ADAPTER EBBusAdapter
  (* Standard: 61499-1 *)
  (* Version 0.0, 2008-04-22, GE, 4DIAC-Consortium *)
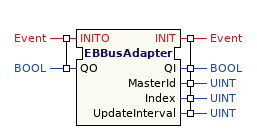
  EVENT_INPUT
    INITO WITH QO; (* Initialization Confirm *)
  END_EVENT
  EVENT_OUTPUT
    INIT WITH Index, UpdateInterval, MasterId, QI; (* Service Initialization *)
  END_EVENT
  VAR_INPUT
    QO : BOOL;
  END_VAR
  VAR_OUTPUT
    QI : BOOL;
    MasterId : UINT;
    Index : UINT;
    UpdateInterval : UINT; (* Global update interval of slave modules in Hz *)
  END_VAR
  SERVICE SOCKET/PLUG
    SEQUENCE request_confirm
      SOCKET.REQ(REQD) -> PLUG.REQ(REQD);
      PLUG.CNF(CNFD) -> SOCKET.CNF(CNFD);
    END_SEQUENCE
    SEQUENCE indication_response
      PLUG.IND(INDD) -> SOCKET.IND(INDD);
      SOCKET.RSP(RSPD) -> PLUG.RSP(RSPD);
    END_SEQUENCE
  END_SERVICE
END_ADAPTER
